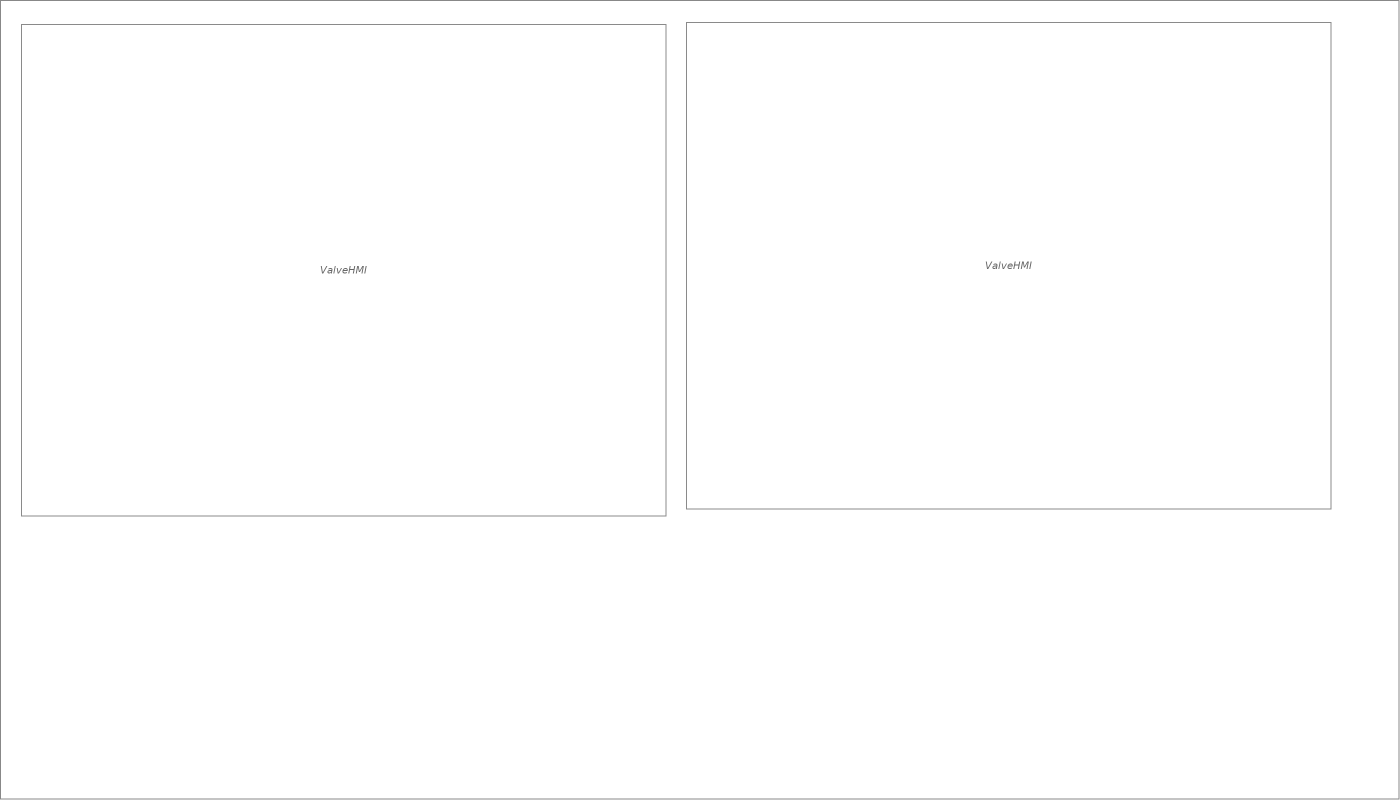
VISUALIZATION Main_Visu  // 1400x800
    Frame (21,24 645x492)
        shows ValveHMI(Valve := GVL_VCM.valve01)
        shows ValveHMI(Valve := GVL_VCM.valve01, ValveIO := GVL_VCM.ioValve01)
    Frame (686,22 645x487)
        shows ValveHMI(Valve := GVL_VCM.valve02, ValveIO := GVL_VCM.ioValve02)
END_VISUALIZATION

(* stored: Version 1.1.0.1, ProductVersion 3.1.4024.12
   Visu Main_Visu: Id {459736cf-f2d9-4d2f-916e-a2ee046ee317} *)
